FUNCTION ForceSetLifterConveyors : BOOL
VAR
	i : INT;
	temp : REFERENCE TO BOOL;
END_VAR

(*
lifter conveyors:
	5..7
	//add more here
*)

FOR i:=5 TO 7 BY 1 DO
	temp REF= allConveyors[i].hasLifter;
	temp := TRUE;
END_FOR

END_FUNCTION

(* stored: Version 1.1.0.1, ProductVersion 3.1.4024.11
   POU ForceSetLifterConveyors: Id {88a3f320-c7c0-4458-aaf6-5a95ff294af9}, SpecialFunc None *)
